FUNCTION_BLOCK FB_PC_OneLink_Cal EXTENDS FB_PC_OneLink_TestSignals
VAR_INPUT
END_VAR
VAR_OUTPUT
END_VAR
VAR
END_VAR


// call the base class to query test signal values
SUPER^();

END_FUNCTION_BLOCK

(* stored: Version 1.1.0.1, ProductVersion 3.1.0.36
   POU FB_PC_OneLink_Cal: Id {b3cdd0c1-f1c6-4a59-a992-429c66a6cb69}, SpecialFunc None *)
